// TIA Portal V20 export
FUNCTION "02 T10 LANT HMI" : Void   // FC1293, LAD
TITLE = HMI
{ S7_Optimized_Access := 'TRUE' }
// stored: AutoNumber false, SetENOAutomatically false
BEGIN

REGION Network 1: Reset command interface from HMI in case of time-out
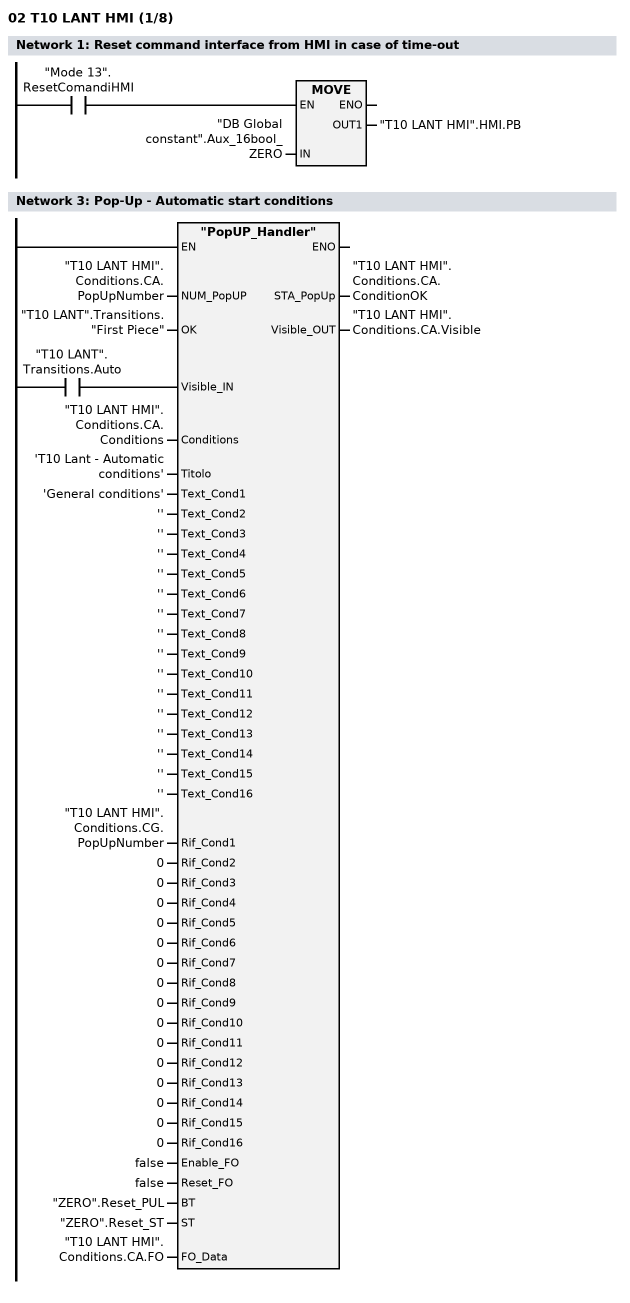
   RUNG wire#powerrail
      Contact( "Mode 13".ResetComandiHMI )
      Move(in := "DB Global constant".Aux_16bool_ZERO, out1 => "T10 LANT HMI".HMI.PB)
   END_RUNG
   // the same network as SCL:
   IF "Mode 13".ResetComandiHMI THEN "T10 LANT HMI".HMI.PB := "DB Global constant".Aux_16bool_ZERO; END_IF;
END_REGION

REGION Network 2: ============ POP UP ============
END_REGION

REGION Network 3: Pop-Up - Automatic start conditions
   RUNG wire#powerrail
      "PopUP_Handler"(Visible_IN := wire#w1, NUM_PopUP := "T10 LANT HMI".Conditions.CA.PopUpNumber, OK := "T10 LANT".Transitions."First Piece", Conditions := "T10 LANT HMI".Conditions.CA.Conditions, Titolo := 'T10 Lant - Automatic conditions', Text_Cond1 := 'General conditions', Text_Cond2 := '', Text_Cond3 := '', Text_Cond4 := '', Text_Cond5 := '', Text_Cond6 := '', Text_Cond7 := '', Text_Cond8 := '', Text_Cond9 := '', Text_Cond10 := '', Text_Cond11 := '', Text_Cond12 := '', Text_Cond13 := '', Text_Cond14 := '', Text_Cond15 := '', Text_Cond16 := '', Rif_Cond1 := "T10 LANT HMI".Conditions.CG.PopUpNumber, Rif_Cond2 := 0, Rif_Cond3 := 0, Rif_Cond4 := 0, Rif_Cond5 := 0, Rif_Cond6 := 0, Rif_Cond7 := 0, Rif_Cond8 := 0, Rif_Cond9 := 0, Rif_Cond10 := 0, Rif_Cond11 := 0, Rif_Cond12 := 0, Rif_Cond13 := 0, Rif_Cond14 := 0, Rif_Cond15 := 0, Rif_Cond16 := 0, Enable_FO := false, Reset_FO := false, BT := "ZERO".Reset_PUL, ST := "ZERO".Reset_ST, FO_Data := "T10 LANT HMI".Conditions.CA.FO, STA_PopUp => "T10 LANT HMI".Conditions.CA.ConditionOK, Visible_OUT => "T10 LANT HMI".Conditions.CA.Visible)
   END_RUNG
   RUNG wire#powerrail
      Contact( "T10 LANT".Transitions.Auto )
   END_RUNG wire#w1
   // the same network as SCL:
   "PopUP_Handler"(NUM_PopUP := "T10 LANT HMI".Conditions.CA.PopUpNumber,
                   OK := "T10 LANT".Transitions."First Piece",
                   Visible_IN := "T10 LANT".Transitions.Auto,
                   Conditions := "T10 LANT HMI".Conditions.CA.Conditions,
                   Titolo := 'T10 Lant - Automatic conditions',
                   Text_Cond1 := 'General conditions',
                   Text_Cond2 := '',
                   Text_Cond3 := '',
                   Text_Cond4 := '',
                   Text_Cond5 := '',
                   Text_Cond6 := '',
                   Text_Cond7 := '',
                   Text_Cond8 := '',
                   Text_Cond9 := '',
                   Text_Cond10 := '',
                   Text_Cond11 := '',
                   Text_Cond12 := '',
                   Text_Cond13 := '',
                   Text_Cond14 := '',
                   Text_Cond15 := '',
                   Text_Cond16 := '',
                   Rif_Cond1 := "T10 LANT HMI".Conditions.CG.PopUpNumber,
                   Rif_Cond2 := 0,
                   Rif_Cond3 := 0,
                   Rif_Cond4 := 0,
                   Rif_Cond5 := 0,
                   Rif_Cond6 := 0,
                   Rif_Cond7 := 0,
                   Rif_Cond8 := 0,
                   Rif_Cond9 := 0,
                   Rif_Cond10 := 0,
                   Rif_Cond11 := 0,
                   Rif_Cond12 := 0,
                   Rif_Cond13 := 0,
                   Rif_Cond14 := 0,
                   Rif_Cond15 := 0,
                   Rif_Cond16 := 0,
                   Enable_FO := false,
                   Reset_FO := false,
                   BT := "ZERO".Reset_PUL,
                   ST := "ZERO".Reset_ST,
                   FO_Data := "T10 LANT HMI".Conditions.CA.FO,
                   STA_PopUp => "T10 LANT HMI".Conditions.CA.ConditionOK,
                   Visible_OUT => "T10 LANT HMI".Conditions.CA.Visible);
END_REGION

REGION Network 4: Pop- Up - General conditions
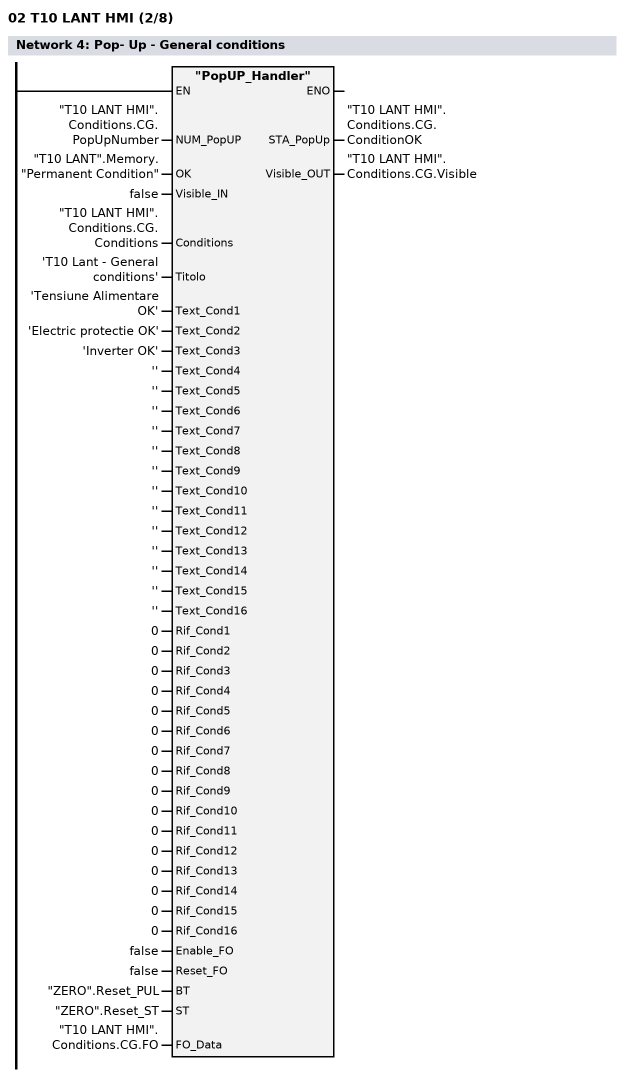
   RUNG wire#powerrail
      "PopUP_Handler"(NUM_PopUP := "T10 LANT HMI".Conditions.CG.PopUpNumber, OK := "T10 LANT".Memory."Permanent Condition", Visible_IN := false, Conditions := "T10 LANT HMI".Conditions.CG.Conditions, Titolo := 'T10 Lant - General conditions', Text_Cond1 := 'Tensiune Alimentare OK', Text_Cond2 := 'Electric protectie OK', Text_Cond3 := 'Inverter OK', Text_Cond4 := '', Text_Cond5 := '', Text_Cond6 := '', Text_Cond7 := '', Text_Cond8 := '', Text_Cond9 := '', Text_Cond10 := '', Text_Cond11 := '', Text_Cond12 := '', Text_Cond13 := '', Text_Cond14 := '', Text_Cond15 := '', Text_Cond16 := '', Rif_Cond1 := 0, Rif_Cond2 := 0, Rif_Cond3 := 0, Rif_Cond4 := 0, Rif_Cond5 := 0, Rif_Cond6 := 0, Rif_Cond7 := 0, Rif_Cond8 := 0, Rif_Cond9 := 0, Rif_Cond10 := 0, Rif_Cond11 := 0, Rif_Cond12 := 0, Rif_Cond13 := 0, Rif_Cond14 := 0, Rif_Cond15 := 0, Rif_Cond16 := 0, Enable_FO := false, Reset_FO := false, BT := "ZERO".Reset_PUL, ST := "ZERO".Reset_ST, FO_Data := "T10 LANT HMI".Conditions.CG.FO, STA_PopUp => "T10 LANT HMI".Conditions.CG.ConditionOK, Visible_OUT => "T10 LANT HMI".Conditions.CG.Visible)
   END_RUNG
   // the same network as SCL:
   "PopUP_Handler"(NUM_PopUP := "T10 LANT HMI".Conditions.CG.PopUpNumber,
                   OK := "T10 LANT".Memory."Permanent Condition",
                   Visible_IN := false,
                   Conditions := "T10 LANT HMI".Conditions.CG.Conditions,
                   Titolo := 'T10 Lant - General conditions',
                   Text_Cond1 := 'Tensiune Alimentare OK',
                   Text_Cond2 := 'Electric protectie OK',
                   Text_Cond3 := 'Inverter OK',
                   Text_Cond4 := '',
                   Text_Cond5 := '',
                   Text_Cond6 := '',
                   Text_Cond7 := '',
                   Text_Cond8 := '',
                   Text_Cond9 := '',
                   Text_Cond10 := '',
                   Text_Cond11 := '',
                   Text_Cond12 := '',
                   Text_Cond13 := '',
                   Text_Cond14 := '',
                   Text_Cond15 := '',
                   Text_Cond16 := '',
                   Rif_Cond1 := 0,
                   Rif_Cond2 := 0,
                   Rif_Cond3 := 0,
                   Rif_Cond4 := 0,
                   Rif_Cond5 := 0,
                   Rif_Cond6 := 0,
                   Rif_Cond7 := 0,
                   Rif_Cond8 := 0,
                   Rif_Cond9 := 0,
                   Rif_Cond10 := 0,
                   Rif_Cond11 := 0,
                   Rif_Cond12 := 0,
                   Rif_Cond13 := 0,
                   Rif_Cond14 := 0,
                   Rif_Cond15 := 0,
                   Rif_Cond16 := 0,
                   Enable_FO := false,
                   Reset_FO := false,
                   BT := "ZERO".Reset_PUL,
                   ST := "ZERO".Reset_ST,
                   FO_Data := "T10 LANT HMI".Conditions.CG.FO,
                   STA_PopUp => "T10 LANT HMI".Conditions.CG.ConditionOK,
                   Visible_OUT => "T10 LANT HMI".Conditions.CG.Visible);
END_REGION

REGION Network 5: PopUP - Cycle start conditions
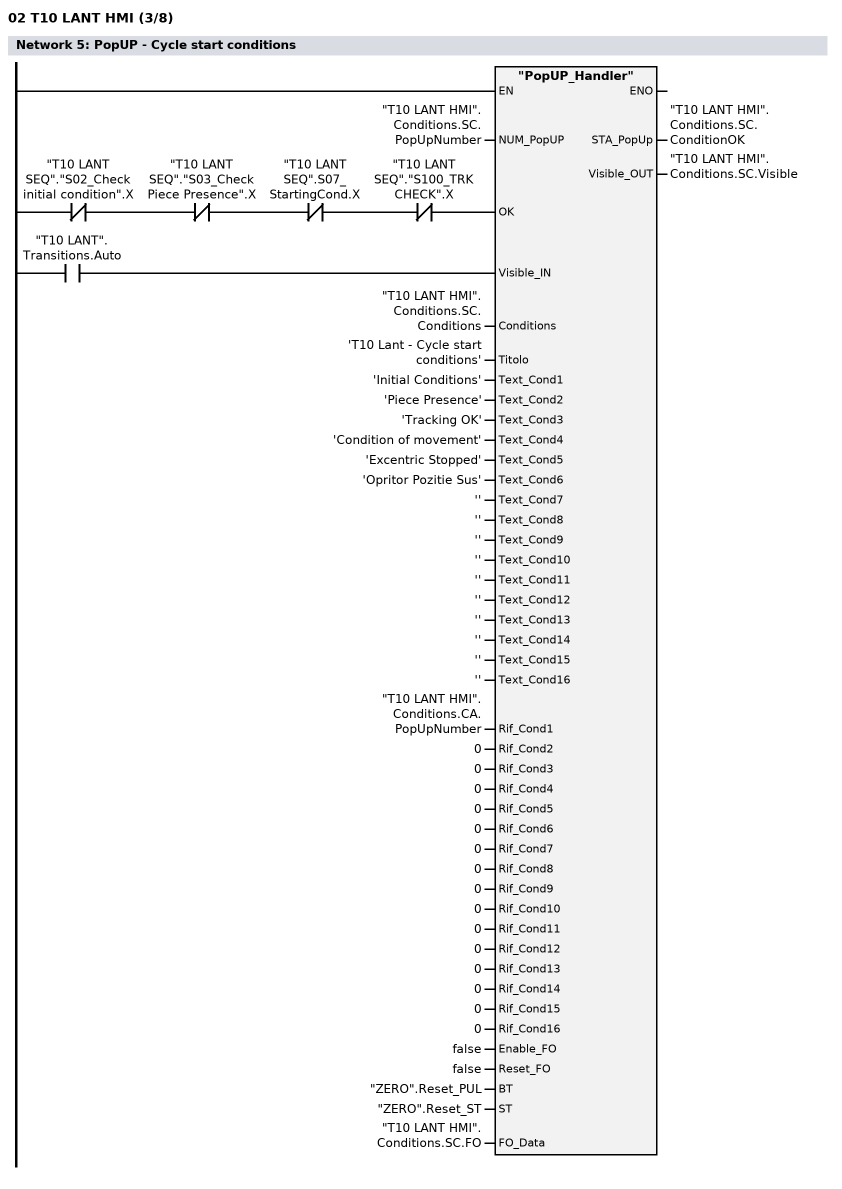
   RUNG wire#powerrail
      "PopUP_Handler"(OK := wire#w1, Visible_IN := wire#w2, NUM_PopUP := "T10 LANT HMI".Conditions.SC.PopUpNumber, Conditions := "T10 LANT HMI".Conditions.SC.Conditions, Titolo := 'T10 Lant - Cycle start conditions', Text_Cond1 := 'Initial Conditions', Text_Cond2 := 'Piece Presence', Text_Cond3 := 'Tracking OK', Text_Cond4 := 'Condition of movement', Text_Cond5 := 'Excentric Stopped', Text_Cond6 := 'Opritor Pozitie Sus', Text_Cond7 := '', Text_Cond8 := '', Text_Cond9 := '', Text_Cond10 := '', Text_Cond11 := '', Text_Cond12 := '', Text_Cond13 := '', Text_Cond14 := '', Text_Cond15 := '', Text_Cond16 := '', Rif_Cond1 := "T10 LANT HMI".Conditions.CA.PopUpNumber, Rif_Cond2 := 0, Rif_Cond3 := 0, Rif_Cond4 := 0, Rif_Cond5 := 0, Rif_Cond6 := 0, Rif_Cond7 := 0, Rif_Cond8 := 0, Rif_Cond9 := 0, Rif_Cond10 := 0, Rif_Cond11 := 0, Rif_Cond12 := 0, Rif_Cond13 := 0, Rif_Cond14 := 0, Rif_Cond15 := 0, Rif_Cond16 := 0, Enable_FO := false, Reset_FO := false, BT := "ZERO".Reset_PUL, ST := "ZERO".Reset_ST, FO_Data := "T10 LANT HMI".Conditions.SC.FO, STA_PopUp => "T10 LANT HMI".Conditions.SC.ConditionOK, Visible_OUT => "T10 LANT HMI".Conditions.SC.Visible)
   END_RUNG
   RUNG wire#powerrail
      I_Contact( "T10 LANT SEQ"."S02_Check initial condition".X )
      I_Contact( "T10 LANT SEQ"."S03_Check Piece Presence".X )
      I_Contact( "T10 LANT SEQ".S07_StartingCond.X )
      I_Contact( "T10 LANT SEQ"."S100_TRK CHECK".X )
   END_RUNG wire#w1
   RUNG wire#powerrail
      Contact( "T10 LANT".Transitions.Auto )
   END_RUNG wire#w2
   // the same network as SCL:
   "PopUP_Handler"(NUM_PopUP := "T10 LANT HMI".Conditions.SC.PopUpNumber,
                   OK := NOT "T10 LANT SEQ"."S02_Check initial condition".X AND NOT "T10 LANT SEQ"."S03_Check Piece Presence".X AND NOT "T10 LANT SEQ".S07_StartingCond.X AND NOT "T10 LANT SEQ"."S100_TRK CHECK".X,
                   Visible_IN := "T10 LANT".Transitions.Auto,
                   Conditions := "T10 LANT HMI".Conditions.SC.Conditions,
                   Titolo := 'T10 Lant - Cycle start conditions',
                   Text_Cond1 := 'Initial Conditions',
                   Text_Cond2 := 'Piece Presence',
                   Text_Cond3 := 'Tracking OK',
                   Text_Cond4 := 'Condition of movement',
                   Text_Cond5 := 'Excentric Stopped',
                   Text_Cond6 := 'Opritor Pozitie Sus',
                   Text_Cond7 := '',
                   Text_Cond8 := '',
                   Text_Cond9 := '',
                   Text_Cond10 := '',
                   Text_Cond11 := '',
                   Text_Cond12 := '',
                   Text_Cond13 := '',
                   Text_Cond14 := '',
                   Text_Cond15 := '',
                   Text_Cond16 := '',
                   Rif_Cond1 := "T10 LANT HMI".Conditions.CA.PopUpNumber,
                   Rif_Cond2 := 0,
                   Rif_Cond3 := 0,
                   Rif_Cond4 := 0,
                   Rif_Cond5 := 0,
                   Rif_Cond6 := 0,
                   Rif_Cond7 := 0,
                   Rif_Cond8 := 0,
                   Rif_Cond9 := 0,
                   Rif_Cond10 := 0,
                   Rif_Cond11 := 0,
                   Rif_Cond12 := 0,
                   Rif_Cond13 := 0,
                   Rif_Cond14 := 0,
                   Rif_Cond15 := 0,
                   Rif_Cond16 := 0,
                   Enable_FO := false,
                   Reset_FO := false,
                   BT := "ZERO".Reset_PUL,
                   ST := "ZERO".Reset_ST,
                   FO_Data := "T10 LANT HMI".Conditions.SC.FO,
                   STA_PopUp => "T10 LANT HMI".Conditions.SC.ConditionOK,
                   Visible_OUT => "T10 LANT HMI".Conditions.SC.Visible);
END_REGION

REGION Network 6: Pop-Up - Conditions of movement FORWARD
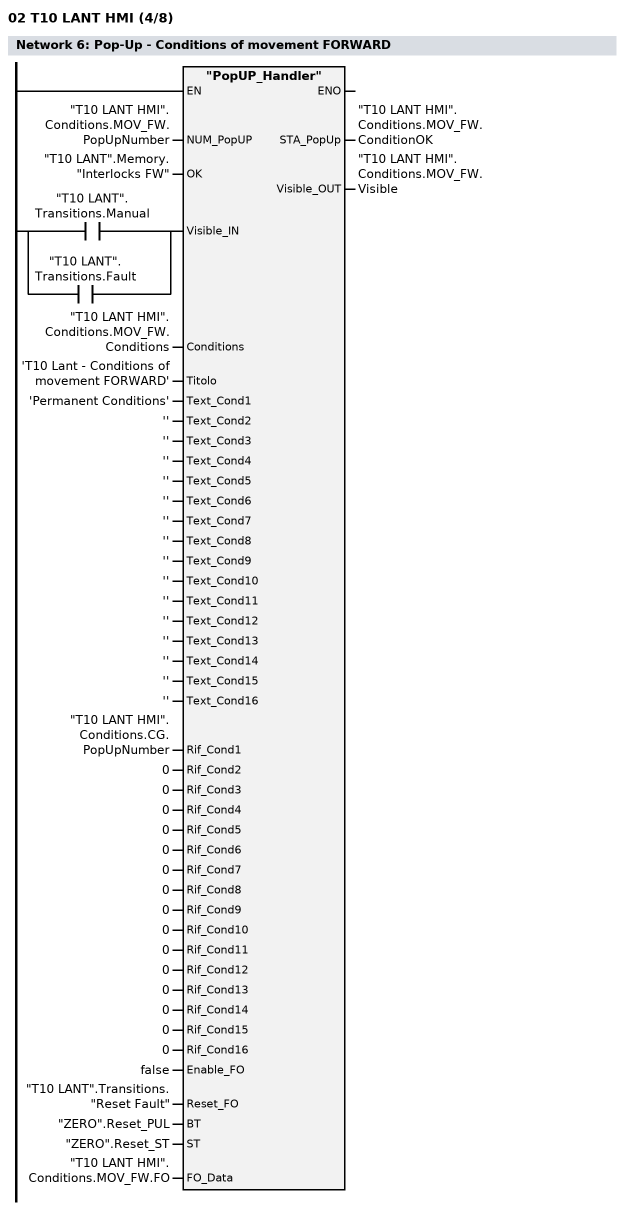
   RUNG wire#powerrail
      "PopUP_Handler"(Visible_IN := wire#w1, NUM_PopUP := "T10 LANT HMI".Conditions.MOV_FW.PopUpNumber, OK := "T10 LANT".Memory."Interlocks FW", Conditions := "T10 LANT HMI".Conditions.MOV_FW.Conditions, Titolo := 'T10 Lant - Conditions of movement FORWARD', Text_Cond1 := 'Permanent Conditions', Text_Cond2 := '', Text_Cond3 := '', Text_Cond4 := '', Text_Cond5 := '', Text_Cond6 := '', Text_Cond7 := '', Text_Cond8 := '', Text_Cond9 := '', Text_Cond10 := '', Text_Cond11 := '', Text_Cond12 := '', Text_Cond13 := '', Text_Cond14 := '', Text_Cond15 := '', Text_Cond16 := '', Rif_Cond1 := "T10 LANT HMI".Conditions.CG.PopUpNumber, Rif_Cond2 := 0, Rif_Cond3 := 0, Rif_Cond4 := 0, Rif_Cond5 := 0, Rif_Cond6 := 0, Rif_Cond7 := 0, Rif_Cond8 := 0, Rif_Cond9 := 0, Rif_Cond10 := 0, Rif_Cond11 := 0, Rif_Cond12 := 0, Rif_Cond13 := 0, Rif_Cond14 := 0, Rif_Cond15 := 0, Rif_Cond16 := 0, Enable_FO := false, Reset_FO := "T10 LANT".Transitions."Reset Fault", BT := "ZERO".Reset_PUL, ST := "ZERO".Reset_ST, FO_Data := "T10 LANT HMI".Conditions.MOV_FW.FO, STA_PopUp => "T10 LANT HMI".Conditions.MOV_FW.ConditionOK, Visible_OUT => "T10 LANT HMI".Conditions.MOV_FW.Visible)
   END_RUNG
   RUNG wire#powerrail
      Contact( "T10 LANT".Transitions.Manual )
   END_RUNG wire#w1
   RUNG wire#powerrail
      Contact( "T10 LANT".Transitions.Fault )
   END_RUNG wire#w1
   // the same network as SCL:
   "PopUP_Handler"(NUM_PopUP := "T10 LANT HMI".Conditions.MOV_FW.PopUpNumber,
                   OK := "T10 LANT".Memory."Interlocks FW",
                   Visible_IN := "T10 LANT".Transitions.Manual OR "T10 LANT".Transitions.Fault,
                   Conditions := "T10 LANT HMI".Conditions.MOV_FW.Conditions,
                   Titolo := 'T10 Lant - Conditions of movement FORWARD',
                   Text_Cond1 := 'Permanent Conditions',
                   Text_Cond2 := '',
                   Text_Cond3 := '',
                   Text_Cond4 := '',
                   Text_Cond5 := '',
                   Text_Cond6 := '',
                   Text_Cond7 := '',
                   Text_Cond8 := '',
                   Text_Cond9 := '',
                   Text_Cond10 := '',
                   Text_Cond11 := '',
                   Text_Cond12 := '',
                   Text_Cond13 := '',
                   Text_Cond14 := '',
                   Text_Cond15 := '',
                   Text_Cond16 := '',
                   Rif_Cond1 := "T10 LANT HMI".Conditions.CG.PopUpNumber,
                   Rif_Cond2 := 0,
                   Rif_Cond3 := 0,
                   Rif_Cond4 := 0,
                   Rif_Cond5 := 0,
                   Rif_Cond6 := 0,
                   Rif_Cond7 := 0,
                   Rif_Cond8 := 0,
                   Rif_Cond9 := 0,
                   Rif_Cond10 := 0,
                   Rif_Cond11 := 0,
                   Rif_Cond12 := 0,
                   Rif_Cond13 := 0,
                   Rif_Cond14 := 0,
                   Rif_Cond15 := 0,
                   Rif_Cond16 := 0,
                   Enable_FO := false,
                   Reset_FO := "T10 LANT".Transitions."Reset Fault",
                   BT := "ZERO".Reset_PUL,
                   ST := "ZERO".Reset_ST,
                   FO_Data := "T10 LANT HMI".Conditions.MOV_FW.FO,
                   STA_PopUp => "T10 LANT HMI".Conditions.MOV_FW.ConditionOK,
                   Visible_OUT => "T10 LANT HMI".Conditions.MOV_FW.Visible);
END_REGION

REGION Network 7: Pop-Up - Conditions of movement BACKWARD
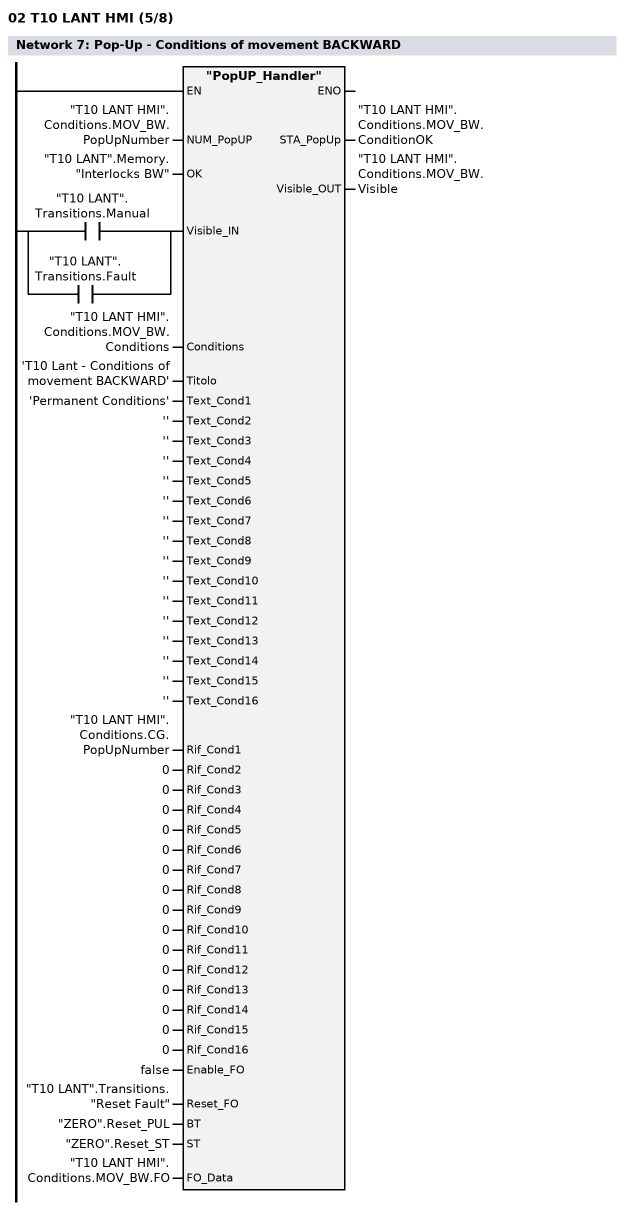
   RUNG wire#powerrail
      "PopUP_Handler"(Visible_IN := wire#w1, NUM_PopUP := "T10 LANT HMI".Conditions.MOV_BW.PopUpNumber, OK := "T10 LANT".Memory."Interlocks BW", Conditions := "T10 LANT HMI".Conditions.MOV_BW.Conditions, Titolo := 'T10 Lant - Conditions of movement BACKWARD', Text_Cond1 := 'Permanent Conditions', Text_Cond2 := '', Text_Cond3 := '', Text_Cond4 := '', Text_Cond5 := '', Text_Cond6 := '', Text_Cond7 := '', Text_Cond8 := '', Text_Cond9 := '', Text_Cond10 := '', Text_Cond11 := '', Text_Cond12 := '', Text_Cond13 := '', Text_Cond14 := '', Text_Cond15 := '', Text_Cond16 := '', Rif_Cond1 := "T10 LANT HMI".Conditions.CG.PopUpNumber, Rif_Cond2 := 0, Rif_Cond3 := 0, Rif_Cond4 := 0, Rif_Cond5 := 0, Rif_Cond6 := 0, Rif_Cond7 := 0, Rif_Cond8 := 0, Rif_Cond9 := 0, Rif_Cond10 := 0, Rif_Cond11 := 0, Rif_Cond12 := 0, Rif_Cond13 := 0, Rif_Cond14 := 0, Rif_Cond15 := 0, Rif_Cond16 := 0, Enable_FO := false, Reset_FO := "T10 LANT".Transitions."Reset Fault", BT := "ZERO".Reset_PUL, ST := "ZERO".Reset_ST, FO_Data := "T10 LANT HMI".Conditions.MOV_BW.FO, STA_PopUp => "T10 LANT HMI".Conditions.MOV_BW.ConditionOK, Visible_OUT => "T10 LANT HMI".Conditions.MOV_BW.Visible)
   END_RUNG
   RUNG wire#powerrail
      Contact( "T10 LANT".Transitions.Manual )
   END_RUNG wire#w1
   RUNG wire#powerrail
      Contact( "T10 LANT".Transitions.Fault )
   END_RUNG wire#w1
   // the same network as SCL:
   "PopUP_Handler"(NUM_PopUP := "T10 LANT HMI".Conditions.MOV_BW.PopUpNumber,
                   OK := "T10 LANT".Memory."Interlocks BW",
                   Visible_IN := "T10 LANT".Transitions.Manual OR "T10 LANT".Transitions.Fault,
                   Conditions := "T10 LANT HMI".Conditions.MOV_BW.Conditions,
                   Titolo := 'T10 Lant - Conditions of movement BACKWARD',
                   Text_Cond1 := 'Permanent Conditions',
                   Text_Cond2 := '',
                   Text_Cond3 := '',
                   Text_Cond4 := '',
                   Text_Cond5 := '',
                   Text_Cond6 := '',
                   Text_Cond7 := '',
                   Text_Cond8 := '',
                   Text_Cond9 := '',
                   Text_Cond10 := '',
                   Text_Cond11 := '',
                   Text_Cond12 := '',
                   Text_Cond13 := '',
                   Text_Cond14 := '',
                   Text_Cond15 := '',
                   Text_Cond16 := '',
                   Rif_Cond1 := "T10 LANT HMI".Conditions.CG.PopUpNumber,
                   Rif_Cond2 := 0,
                   Rif_Cond3 := 0,
                   Rif_Cond4 := 0,
                   Rif_Cond5 := 0,
                   Rif_Cond6 := 0,
                   Rif_Cond7 := 0,
                   Rif_Cond8 := 0,
                   Rif_Cond9 := 0,
                   Rif_Cond10 := 0,
                   Rif_Cond11 := 0,
                   Rif_Cond12 := 0,
                   Rif_Cond13 := 0,
                   Rif_Cond14 := 0,
                   Rif_Cond15 := 0,
                   Rif_Cond16 := 0,
                   Enable_FO := false,
                   Reset_FO := "T10 LANT".Transitions."Reset Fault",
                   BT := "ZERO".Reset_PUL,
                   ST := "ZERO".Reset_ST,
                   FO_Data := "T10 LANT HMI".Conditions.MOV_BW.FO,
                   STA_PopUp => "T10 LANT HMI".Conditions.MOV_BW.ConditionOK,
                   Visible_OUT => "T10 LANT HMI".Conditions.MOV_BW.Visible);
END_REGION

REGION Network 8: ============ HMI STATE ============
END_REGION

REGION Network 9: HMI Status - Commands
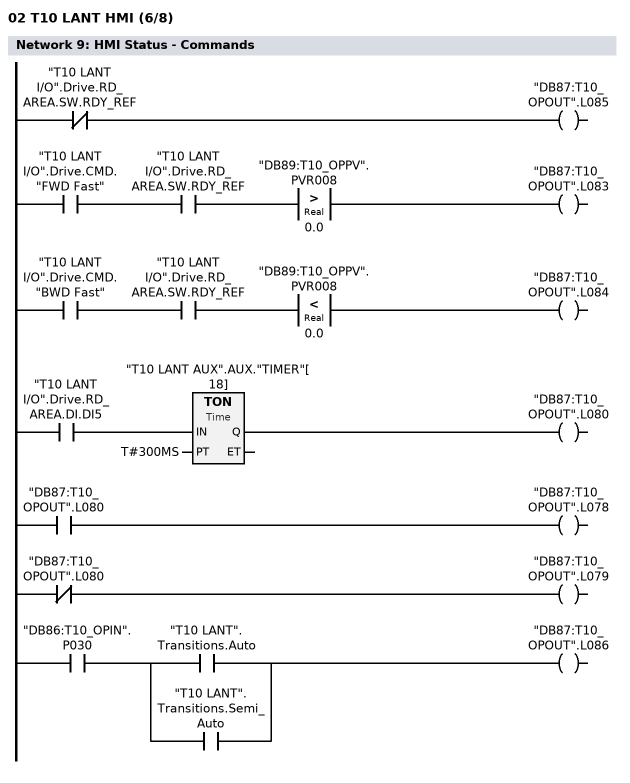
   RUNG wire#powerrail
      I_Contact( "T10 LANT I/O".Drive.RD_AREA.SW.RDY_REF )
      Coil( "DB87:T10_OPOUT".L085 )
   END_RUNG
   RUNG wire#powerrail
      Contact( "T10 LANT I/O".Drive.CMD."FWD Fast" )
      Contact( "T10 LANT I/O".Drive.RD_AREA.SW.RDY_REF )
      { S7_Templates := "SrcType := Real" } GT_Contact(in1 := "DB89:T10_OPPV".PVR008, in2 := 0.0)
      Coil( "DB87:T10_OPOUT".L083 )
   END_RUNG
   RUNG wire#powerrail
      Contact( "T10 LANT I/O".Drive.CMD."BWD Fast" )
      Contact( "T10 LANT I/O".Drive.RD_AREA.SW.RDY_REF )
      { S7_Templates := "SrcType := Real" } LT_Contact(in1 := "DB89:T10_OPPV".PVR008, in2 := 0.0)
      Coil( "DB87:T10_OPOUT".L084 )
   END_RUNG
   RUNG wire#powerrail
      Contact( "T10 LANT I/O".Drive.RD_AREA.DI.DI5 )
      { S7_Templates := "time_type := Time" } "T10 LANT AUX".AUX."TIMER"[18].TON(pt := T#300MS, et =>)
      Coil( "DB87:T10_OPOUT".L080 )
   END_RUNG
   RUNG wire#powerrail
      Contact( "DB87:T10_OPOUT".L080 )
      Coil( "DB87:T10_OPOUT".L078 )
   END_RUNG
   RUNG wire#powerrail
      I_Contact( "DB87:T10_OPOUT".L080 )
      Coil( "DB87:T10_OPOUT".L079 )
   END_RUNG
   RUNG wire#powerrail
      Contact( "DB86:T10_OPIN".P030 )
      wire#w1
      Contact( "T10 LANT".Transitions.Auto )
      wire#w2
      Coil( "DB87:T10_OPOUT".L086 )
   END_RUNG
   RUNG wire#w1
      Contact( "T10 LANT".Transitions.Semi_Auto )
   END_RUNG wire#w2
   // the same network as SCL:
   "DB87:T10_OPOUT".L085 := NOT "T10 LANT I/O".Drive.RD_AREA.SW.RDY_REF;
   "DB87:T10_OPOUT".L083 := "T10 LANT I/O".Drive.CMD."FWD Fast" AND "T10 LANT I/O".Drive.RD_AREA.SW.RDY_REF AND ("DB89:T10_OPPV".PVR008 > 0.0);
   "DB87:T10_OPOUT".L084 := "T10 LANT I/O".Drive.CMD."BWD Fast" AND "T10 LANT I/O".Drive.RD_AREA.SW.RDY_REF AND ("DB89:T10_OPPV".PVR008 < 0.0);
   "T10 LANT AUX".AUX."TIMER"[18].TON(IN := "T10 LANT I/O".Drive.RD_AREA.DI.DI5, PT := T#300MS);
   "DB87:T10_OPOUT".L080 := "T10 LANT AUX".AUX."TIMER"[18].Q;
   "DB87:T10_OPOUT".L078 := "DB87:T10_OPOUT".L080;
   "DB87:T10_OPOUT".L079 := NOT "DB87:T10_OPOUT".L080;
   "DB87:T10_OPOUT".L086 := "DB86:T10_OPIN".P030 AND ("T10 LANT".Transitions.Auto OR "T10 LANT".Transitions.Semi_Auto);
END_REGION

REGION Network 10: HMI Status - Sensors
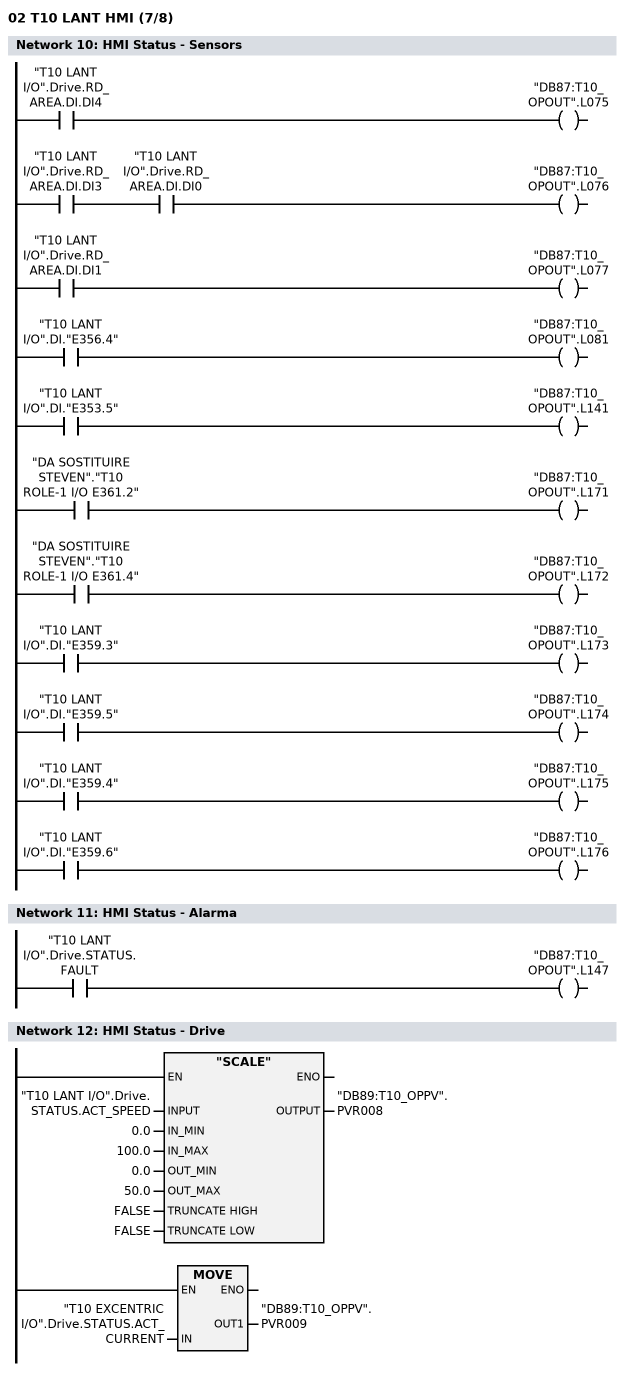
   RUNG wire#powerrail
      Contact( "T10 LANT I/O".Drive.RD_AREA.DI.DI4 )
      Coil( "DB87:T10_OPOUT".L075 )
   END_RUNG
   RUNG wire#powerrail
      Contact( "T10 LANT I/O".Drive.RD_AREA.DI.DI3 )
      Contact( "T10 LANT I/O".Drive.RD_AREA.DI.DI0 )
      Coil( "DB87:T10_OPOUT".L076 )
   END_RUNG
   RUNG wire#powerrail
      Contact( "T10 LANT I/O".Drive.RD_AREA.DI.DI1 )
      Coil( "DB87:T10_OPOUT".L077 )
   END_RUNG
   RUNG wire#powerrail
      Contact( "T10 LANT I/O".DI."E356.4" )
      Coil( "DB87:T10_OPOUT".L081 )
   END_RUNG
   RUNG wire#powerrail
      Contact( "T10 LANT I/O".DI."E353.5" )
      Coil( "DB87:T10_OPOUT".L141 )
   END_RUNG
   RUNG wire#powerrail
      Contact( "DA SOSTITUIRE STEVEN"."T10 ROLE-1 I/O E361.2" )
      Coil( "DB87:T10_OPOUT".L171 )
   END_RUNG
   RUNG wire#powerrail
      Contact( "DA SOSTITUIRE STEVEN"."T10 ROLE-1 I/O E361.4" )
      Coil( "DB87:T10_OPOUT".L172 )
   END_RUNG
   RUNG wire#powerrail
      Contact( "T10 LANT I/O".DI."E359.3" )
      Coil( "DB87:T10_OPOUT".L173 )
   END_RUNG
   RUNG wire#powerrail
      Contact( "T10 LANT I/O".DI."E359.5" )
      Coil( "DB87:T10_OPOUT".L174 )
   END_RUNG
   RUNG wire#powerrail
      Contact( "T10 LANT I/O".DI."E359.4" )
      Coil( "DB87:T10_OPOUT".L175 )
   END_RUNG
   RUNG wire#powerrail
      Contact( "T10 LANT I/O".DI."E359.6" )
      Coil( "DB87:T10_OPOUT".L176 )
   END_RUNG
   // the same network as SCL:
   "DB87:T10_OPOUT".L075 := "T10 LANT I/O".Drive.RD_AREA.DI.DI4;
   "DB87:T10_OPOUT".L076 := "T10 LANT I/O".Drive.RD_AREA.DI.DI3 AND "T10 LANT I/O".Drive.RD_AREA.DI.DI0;
   "DB87:T10_OPOUT".L077 := "T10 LANT I/O".Drive.RD_AREA.DI.DI1;
   "DB87:T10_OPOUT".L081 := "T10 LANT I/O".DI."E356.4";
   "DB87:T10_OPOUT".L141 := "T10 LANT I/O".DI."E353.5";
   "DB87:T10_OPOUT".L171 := "DA SOSTITUIRE STEVEN"."T10 ROLE-1 I/O E361.2";
   "DB87:T10_OPOUT".L172 := "DA SOSTITUIRE STEVEN"."T10 ROLE-1 I/O E361.4";
   "DB87:T10_OPOUT".L173 := "T10 LANT I/O".DI."E359.3";
   "DB87:T10_OPOUT".L174 := "T10 LANT I/O".DI."E359.5";
   "DB87:T10_OPOUT".L175 := "T10 LANT I/O".DI."E359.4";
   "DB87:T10_OPOUT".L176 := "T10 LANT I/O".DI."E359.6";
END_REGION

REGION Network 11: HMI Status - Alarma
   RUNG wire#powerrail
      Contact( "T10 LANT I/O".Drive.STATUS.FAULT )
      Coil( "DB87:T10_OPOUT".L147 )
   END_RUNG
   // the same network as SCL:
   "DB87:T10_OPOUT".L147 := "T10 LANT I/O".Drive.STATUS.FAULT;
END_REGION

REGION Network 12: HMI Status - Drive
   RUNG wire#powerrail
      "SCALE"(INPUT := "T10 LANT I/O".Drive.STATUS.ACT_SPEED, IN_MIN := 0.0, IN_MAX := 100.0, OUT_MIN := 0.0, OUT_MAX := 50.0, "TRUNCATE HIGH" := FALSE, "TRUNCATE LOW" := FALSE, OUTPUT => "DB89:T10_OPPV".PVR008)
   END_RUNG
   RUNG wire#powerrail
      Move(in := "T10 EXCENTRIC I/O".Drive.STATUS.ACT_CURRENT, out1 => "DB89:T10_OPPV".PVR009)
   END_RUNG
   // the same network as SCL:
   "SCALE"(INPUT := "T10 LANT I/O".Drive.STATUS.ACT_SPEED,
           IN_MIN := 0.0,
           IN_MAX := 100.0,
           OUT_MIN := 0.0,
           OUT_MAX := 50.0,
           "TRUNCATE HIGH" := FALSE,
           "TRUNCATE LOW" := FALSE,
           OUTPUT => "DB89:T10_OPPV".PVR008);
   "DB89:T10_OPPV".PVR009 := "T10 EXCENTRIC I/O".Drive.STATUS.ACT_CURRENT;
END_REGION

REGION Network 13: Device status
   // m0.7 comandi uscite
   // M0.7 minimun energy conditions
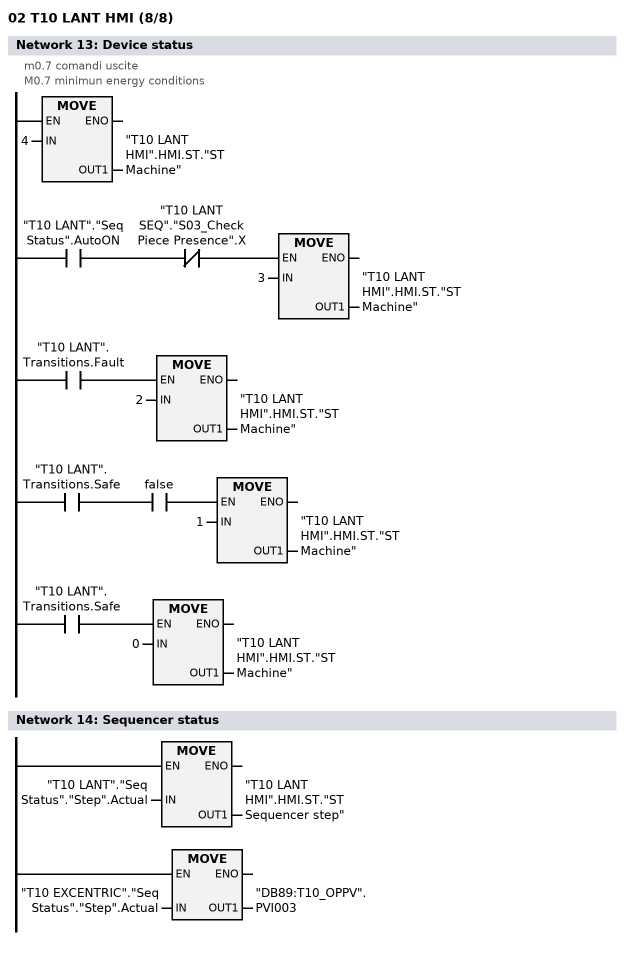
   RUNG wire#powerrail
      Move(in := 4, out1 => "T10 LANT HMI".HMI.ST."ST Machine")
   END_RUNG
   RUNG wire#powerrail
      Contact( "T10 LANT"."Seq Status".AutoON )
      I_Contact( "T10 LANT SEQ"."S03_Check Piece Presence".X )
      Move(in := 3, out1 => "T10 LANT HMI".HMI.ST."ST Machine")
   END_RUNG
   RUNG wire#powerrail
      Contact( "T10 LANT".Transitions.Fault )
      Move(in := 2, out1 => "T10 LANT HMI".HMI.ST."ST Machine")
   END_RUNG
   RUNG wire#powerrail
      Contact( "T10 LANT".Transitions.Safe )
      Contact( false )
      Move(in := 1, out1 => "T10 LANT HMI".HMI.ST."ST Machine")
   END_RUNG
   RUNG wire#powerrail
      Contact( "T10 LANT".Transitions.Safe )
      Move(in := 0, out1 => "T10 LANT HMI".HMI.ST."ST Machine")
   END_RUNG
   // the same network as SCL:
   "T10 LANT HMI".HMI.ST."ST Machine" := 4;
   IF "T10 LANT"."Seq Status".AutoON AND NOT "T10 LANT SEQ"."S03_Check Piece Presence".X THEN
       "T10 LANT HMI".HMI.ST."ST Machine" := 3;
   END_IF;
   IF "T10 LANT".Transitions.Fault THEN "T10 LANT HMI".HMI.ST."ST Machine" := 2; END_IF;
   IF "T10 LANT".Transitions.Safe AND false THEN "T10 LANT HMI".HMI.ST."ST Machine" := 1; END_IF;
   IF "T10 LANT".Transitions.Safe THEN "T10 LANT HMI".HMI.ST."ST Machine" := 0; END_IF;
END_REGION

REGION Network 14: Sequencer status
   RUNG wire#powerrail
      Move(in := "T10 LANT"."Seq Status"."Step".Actual, out1 => "T10 LANT HMI".HMI.ST."ST Sequencer step")
   END_RUNG
   RUNG wire#powerrail
      Move(in := "T10 EXCENTRIC"."Seq Status"."Step".Actual, out1 => "DB89:T10_OPPV".PVI003)
   END_RUNG
   // the same network as SCL:
   "T10 LANT HMI".HMI.ST."ST Sequencer step" := "T10 LANT"."Seq Status"."Step".Actual;
   "DB89:T10_OPPV".PVI003 := "T10 EXCENTRIC"."Seq Status"."Step".Actual;
END_REGION
END_FUNCTION
